// TIA Portal V19 export
VAR_GLOBAL   // PLC tag table "Equipment_Template_DefaultTagTable_5"
   "Tag_49(2)" AT %I30142.0 : Bool;   // 物流线允许出
   "Tag_50(2)" AT %I30142.1 : Bool;   // 物流线通知托盘送出完成
   "Tag_51(2)" AT %I30142.2 : Bool;   // 物流线收到单机收到的物流线出到位信号
   "Tag_52(2)" AT %I30142.3 : Bool;   // 物流线空闲
   "Tag_53(2)" AT %I30142.4 : Bool;
   "Tag_54(2)" AT %I30142.5 : Bool;
   "Tag_55(2)" AT %I30142.6 : Bool;
   "Tag_56(2)" AT %I30142.7 : Bool;   // 物流请求出托盘
   "Tag_57(2)" AT %I30143.0 : Bool;   // 物流线忙碌
   "Tag_58(2)" AT %I30143.1 : Bool;   // 物流线收到单机返回出到位信号
   "Tag_59(2)" AT %I30143.2 : Bool;   // 物流工位报警
   "Tag_60(2)" AT %I30143.3 : Bool;   // 物流有拖盘待出
   "Tag_61(2)" AT %I30143.4 : Bool;
   "Tag_62(2)" AT %I30143.5 : Bool;
   "Tag_63(2)" AT %I30143.6 : Bool;
   "Tag_64(2)" AT %I30143.7 : Bool;
END_VAR
